// TIA Portal V18 program export: 1 tag tables, 0 data types, 0 data blocks, 6 code blocks (in call order from the OBs), 0 instance data blocks

VAR_GLOBAL   // PLC tag table "Default tag table"
   convRight AT %I0.0 : Bool;
   convLeft AT %I0.1 : Bool;
   manualMode AT %Q0.2 : Bool;
   automaticMode AT %Q0.3 : Bool;
END_VAR

ORGANIZATION_BLOCK "Main"   // OB1, LAD, ProgramCycle
TITLE = "Main Program Sweep (Cycle)"
{ S7_Optimized_Access := 'TRUE' }
VERSION : 0.1
// stored: AutoNumber true, IsIECCheckEnabled true, SetENOAutomatically false
   VAR_INPUT
      Initial_Call : Bool;   // Initial call of this OB
      Remanence : Bool;   // =True, if remanent data are available
   END_VAR
BEGIN
END_ORGANIZATION_BLOCK

FUNCTION_BLOCK "Conveyor"   // FB2, FBD
{ S7_Optimized_Access := 'TRUE' }
AUTHOR : dda
VERSION : 0.1
// stored: AutoNumber true, IsIECCheckEnabled true, IsRetainMemResEnabled false, MemoryReserve 100, SetENOAutomatically true, UDAEnableTagReadback false
   VAR_INPUT
      automaticMode { ExternalAccessible := 'False'; ExternalVisible := 'False'; ExternalWritable := 'False'} : Bool;
      manualMode { ExternalAccessible := 'False'; ExternalVisible := 'False'; ExternalWritable := 'False'} : Bool;
      jogRight { ExternalAccessible := 'False'; ExternalVisible := 'False'; ExternalWritable := 'False'} : Bool;
      run { ExternalAccessible := 'False'; ExternalVisible := 'False'; ExternalWritable := 'False'} : Bool;
   END_VAR
   VAR_OUTPUT
      conveyorRight { ExternalAccessible := 'False'; ExternalVisible := 'False'; ExternalWritable := 'False'} : Bool;
      conveyorLeft { ExternalAccessible := 'False'; ExternalVisible := 'False'; ExternalWritable := 'False'} : Bool;
   END_VAR
   VAR
      statRequest { ExternalAccessible := 'False'; ExternalVisible := 'False'; ExternalWritable := 'False'} : Bool;
      statRelease { ExternalAccessible := 'False'; ExternalVisible := 'False'; ExternalWritable := 'False'} : Bool;
   END_VAR
BEGIN

REGION Network 1 (SCL)
   // functionality: conveyor
   //
END_REGION

REGION Network 2
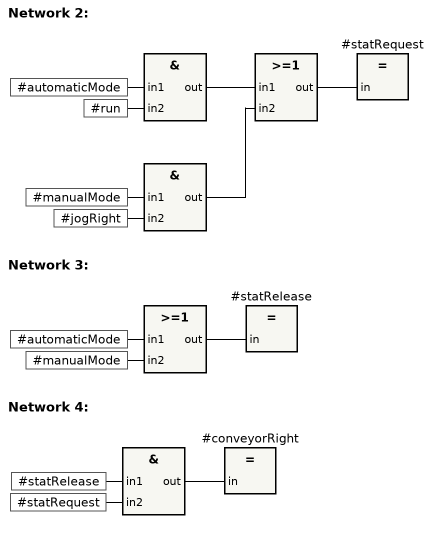
   #statRequest := (#automaticMode AND #run) OR (#manualMode AND #jogRight);
END_REGION

REGION Network 3
   #statRelease := #automaticMode OR #manualMode;
END_REGION

REGION Network 4
   #conveyorRight := #statRelease AND #statRequest;
END_REGION
END_FUNCTION_BLOCK

FUNCTION_BLOCK "Seqencer"   // FB4, GRAPH
AUTHOR : dda
VERSION : 0.1
// stored: AcknowledgeErrorsRequired true, AutoNumber true, GraphVersion 6.0, InitialValuesAcquisition false, IsIECCheckEnabled true, LanguageInNetworks FBD, LockOperatingMode false, PermanentILProcessingInMANMode false, SetENOAutomatically true, SkipSteps false, UDAEnableTagReadback false, WithAlarmHandling true
   // inherited from GRAPH_BASE
   VAR
      OFF_SQ_BASE : Bool;
   END_VAR
   VAR_INPUT
      OFF_SQ { ExternalWritable := 'False'} : Bool := false;   // Turn sequence off
      INIT_SQ { ExternalWritable := 'False'} : Bool := false;   // Set sequence to initial state
      ACK_EF { ExternalWritable := 'False'} : Bool := false;   // Acknowledge all errors and faults
      REG_EF { ExternalWritable := 'False'} : Bool := false;   // Register all errors and faults
      ACK_S { ExternalWritable := 'False'} : Bool := false;   // Acknowledge step indicated in S_NO
      REG_S { ExternalWritable := 'False'} : Bool := false;   // Register the step indicated in S_NO
      HALT_SQ { ExternalWritable := 'False'} : Bool := false;   // Halt sequence immediately
      HALT_TM { ExternalWritable := 'False'} : Bool := false;   // Halt timers immediately
      ZERO_OP { ExternalWritable := 'False'} : Bool := false;   // Set all operands assigned with N, L, D to 0
      EN_IL { ExternalWritable := 'False'} : Bool := false;   // Enable interlocks
      EN_SV { ExternalWritable := 'False'} : Bool := false;   // Activate supervision processing
      EN_ACKREQ { ExternalWritable := 'False'} : Bool := false;   // Activate mandatory acknowledgment
      EN_SSKIP { ExternalWritable := 'False'} : Bool := false;   // Enable "Skip step"
      DISP_SACT { ExternalWritable := 'False'} : Bool := false;   // Display active steps only
      DISP_SEF { ExternalWritable := 'False'} : Bool := false;   // Display only steps with errors and disrupted steps
      DISP_SALL { ExternalWritable := 'False'} : Bool := false;   // Display all steps
      S_PREV { ExternalWritable := 'False'} : Bool := false;   // Output previous step in parameter S_NO
      S_NEXT { ExternalWritable := 'False'} : Bool := false;   // Indicate next step in parameter S_NO
      SW_AUTO { ExternalWritable := 'False'} : Bool := false;   // Automatic mode
      SW_TAP { ExternalWritable := 'False'} : Bool := false;   // Semiautomatic/switch with transition
      SW_TOP { ExternalWritable := 'False'} : Bool := false;   // Semiautomatic/ignore transition
      SW_MAN { ExternalWritable := 'False'} : Bool := false;   // Manual mode
      S_SEL { ExternalWritable := 'False'} : Int := 0;   // Select step to be output to S_NO
      S_SELOK { ExternalWritable := 'False'} : Bool := false;   // Enter value from S_SEL in S_NO
      S_ON { ExternalWritable := 'False'} : Bool := false;   // Activate step indicated in S_NO
      S_OFF { ExternalWritable := 'False'} : Bool := false;   // Disable step indicated in S_NO
      T_PREV { ExternalWritable := 'False'} : Bool := false;   // Display previous transition in T_NO
      T_NEXT { ExternalWritable := 'False'} : Bool := false;   // Display next transition at parameter T_NO
      T_PUSH { ExternalWritable := 'False'} : Bool := false;   // Enable transition to switch in semi automatic mode
      EN_LMODE { ExternalWritable := 'False'} : Bool := false;   // Activate learning mode
      RESET_CRIT { ExternalWritable := 'False'} : Bool := false;   // Reset all initial values recorded for interlocks and transitions
      startButton : Bool;
      lightBeam1 : Bool;
      lightBeam2 : Bool;
      lightBeam3 : Bool;
      robotArmDown : Bool;
      robotOnStation : Bool;
      robotOnMagazine : Bool;
      mySupervision : Bool;
   END_VAR
   VAR_OUTPUT
      S_NO { ExternalWritable := 'False'} : Int := 0;   // Step number
      S_MORE { ExternalWritable := 'False'} : Bool := false;   // More steps are available and can be shown in S_NO
      S_ACTIVE { ExternalWritable := 'False'} : Bool := false;   // Step indicated in S_NO is active
      S_TIME { ExternalWritable := 'False'} : Time := T#0ms;   // Step activation time
      S_TIMEOK { ExternalWritable := 'False'} : Time := T#0ms;   // No error in step activation time
      S_CRITLOC { ExternalWritable := 'False'} : DWord := 16#0;   // Interlock criteria bits
      S_CRITLOCERR { ExternalWritable := 'False'} : DWord := 16#0;   // Interlock criteria bits for event L1
      S_STATE { ExternalWritable := 'False'} : Word := 16#0;   // Step state bits
      T_NO { ExternalWritable := 'False'} : Int := 0;   // Transition number
      T_MORE { ExternalWritable := 'False'} : Bool := false;   // More valid transitions available for display
      T_CRIT { ExternalWritable := 'False'} : DWord := 16#0;   // Transition criteria bits
      T_CRITOLD { ExternalWritable := 'False'} : DWord := 16#0;   // Transition criteria bits from last cycle
      T_CRITFLT { ExternalWritable := 'False'} : DWord := 16#0;   // Transition criteria bits for event V1
      ERROR { ExternalWritable := 'False'} : Bool := false;   // Interlock group error
      FAULT { ExternalWritable := 'False'} : Bool := false;   // Supervision group error
      ERR_FLT { ExternalWritable := 'False'} : Bool := false;   // Interlock or supervision group error
      SQ_ISOFF { ExternalWritable := 'False'} : Bool := false;   // Sequence is off (no step active)
      SQ_HALTED { ExternalWritable := 'False'} : Bool := false;   // Sequence halted
      TM_HALTED { ExternalWritable := 'False'} : Bool := false;   // Timers halted
      OP_ZEROED { ExternalWritable := 'False'} : Bool := false;   // All the operands assigned with N, L, D are set to 0
      IL_ENABLED { ExternalWritable := 'False'} : Bool := false;   // Interlocks are active
      SV_ENABLED { ExternalWritable := 'False'} : Bool := false;   // Supervision processing activated
      ACKREQ_ENABLED { ExternalWritable := 'False'} : Bool := false;   // Mandatory acknowledgment activated
      SSKIP_ENABLED { ExternalWritable := 'False'} : Bool := false;   // Skip steps activated
      SACT_DISP { ExternalWritable := 'False'} : Bool := false;   // Display active steps only
      SEF_DISP { ExternalWritable := 'False'} : Bool := false;   // Display only steps with errors or disrupted steps
      SALL_DISP { ExternalWritable := 'False'} : Bool := false;   // Display all steps
      AUTO_ON { ExternalWritable := 'False'} : Bool := false;   // Automatic mode is active
      TAP_ON { ExternalWritable := 'False'} : Bool := false;   // Semiautomatic mode/step with transition enabled
      TOP_ON { ExternalWritable := 'False'} : Bool := false;   // Semiautomatic mode/ignore transition enabled
      MAN_ON { ExternalWritable := 'False'} : Bool := false;   // Manual mode is active
      LMODE_ENABLED { ExternalWritable := 'False'} : Bool := false;   // Learning mode is active
      partInPos1 { ExternalAccessible := 'False'; ExternalVisible := 'False'; ExternalWritable := 'False'} : Bool;
      partInPos2 { ExternalAccessible := 'False'; ExternalVisible := 'False'; ExternalWritable := 'False'} : Bool;
      partInPos3 { ExternalAccessible := 'False'; ExternalVisible := 'False'; ExternalWritable := 'False'} : Bool;
      startConv { ExternalAccessible := 'False'; ExternalVisible := 'False'; ExternalWritable := 'False'} : Bool;
      automaticMode { ExternalAccessible := 'False'; ExternalVisible := 'False'; ExternalWritable := 'False'} : Bool;
      robotFill { ExternalAccessible := 'False'; ExternalVisible := 'False'; ExternalWritable := 'False'} : Bool;
      robotGoToMagazine { ExternalAccessible := 'False'; ExternalVisible := 'False'; ExternalWritable := 'False'} : Bool;
      robotGoToStation { ExternalAccessible := 'False'; ExternalVisible := 'False'; ExternalWritable := 'False'} : Bool;
   END_VAR
   VAR
      statLightbeam3Fal { ExternalAccessible := 'False'; ExternalVisible := 'False'; ExternalWritable := 'False'} : Bool;
      statMemoryTag { ExternalAccessible := 'False'; ExternalVisible := 'False'; ExternalWritable := 'False'} : Bool;
   END_VAR
BEGIN
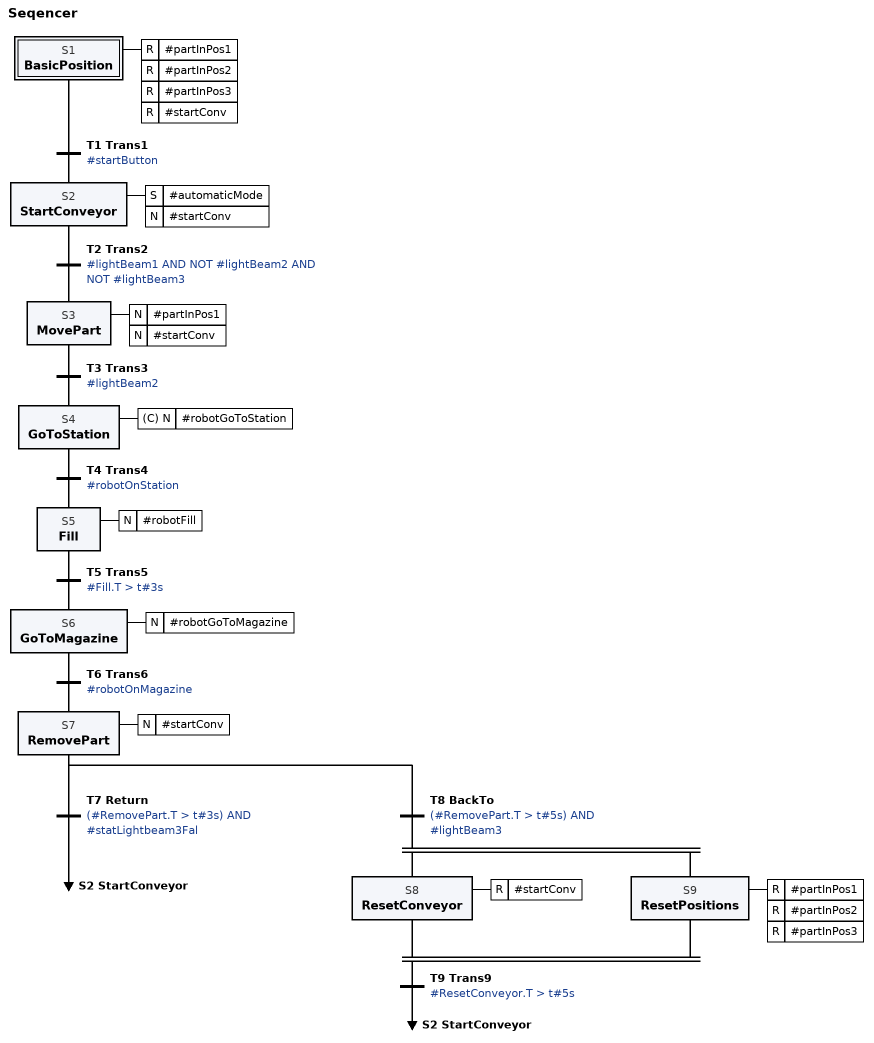
   // sequencer 1
   INITIAL_STEP BasicPosition:   // S1, max time T#10S, warning time T#7S
      supervision V := (#StartConveyor.T > t#10ms) AND (#StartConveyor.U > t#10ms);
              R    #partInPos1
              R    #partInPos2
              R    #partInPos3
              R    #startConv
   END_STEP
   TRANSITION Trans1 FROM BasicPosition TO StartConveyor   // T1
      := #startButton;
   END_TRANSITION
   STEP StartConveyor:   // S2, max time T#10S, warning time T#7S
              S    #automaticMode
              N    #startConv
   END_STEP
   TRANSITION Trans2 FROM StartConveyor TO MovePart   // T2
      := #lightBeam1 AND NOT #lightBeam2 AND NOT #lightBeam3;
   END_TRANSITION
   STEP MovePart:   // S3, max time T#10S, warning time T#7S
              N    #partInPos1
              N    #startConv
   END_STEP
   TRANSITION Trans3 FROM MovePart TO GoToStation   // T3
      := #lightBeam2;
   END_TRANSITION
   STEP GoToStation:   // S4, max time T#10S, warning time T#7S
      interlock C := NOT #robotArmDown;
      (C)     N    #robotGoToStation
   END_STEP
   TRANSITION Trans4 FROM GoToStation TO Fill   // T4
      := #robotOnStation;
   END_TRANSITION
   STEP Fill:   // S5, max time T#10S, warning time T#7S
              N    #robotFill
   END_STEP
   TRANSITION Trans5 FROM Fill TO GoToMagazine   // T5
      := #Fill.T > t#3s;
   END_TRANSITION
   STEP GoToMagazine:   // S6, max time T#10S, warning time T#7S
              N    #robotGoToMagazine
   END_STEP
   TRANSITION Trans6 FROM GoToMagazine TO RemovePart   // T6
      := #robotOnMagazine;
   END_TRANSITION
   STEP RemovePart:   // S7, max time T#10S, warning time T#7S
      supervision V := (#RemovePart.T < #RemovePart.T_MAX) AND (#RemovePart.T > #RemovePart.T_WARN);
              N    #startConv
   END_STEP
   TRANSITION "Return" FROM RemovePart TO StartConveyor   // T7, jump
      := (#RemovePart.T > t#3s) AND #statLightbeam3Fal;
   END_TRANSITION
   TRANSITION BackTo FROM RemovePart TO (ResetConveyor, ResetPositions)   // T8
      := (#RemovePart.T > t#5s) AND #lightBeam3;
   END_TRANSITION
   STEP ResetConveyor:   // S8, max time T#10S, warning time T#7S
              R    #startConv
   END_STEP
   STEP ResetPositions:   // S9, max time T#10S, warning time T#7S
      interlock C := #ResetPositions.T > #ResetPositions.T_MAX;
              R    #partInPos1
              R    #partInPos2
              R    #partInPos3
   END_STEP
   TRANSITION Trans9 FROM (ResetConveyor, ResetPositions) TO StartConveyor   // T9, jump
      := #ResetConveyor.T > t#5s;
   END_TRANSITION
END_FUNCTION_BLOCK

FUNCTION_BLOCK "Simulation"   // FB1, FBD
TITLE = Simulation
{ S7_Optimized_Access := 'TRUE' }
AUTHOR : dda
VERSION : 0.1
// Simulate machine behaviour
// stored: AutoNumber true, IsIECCheckEnabled true, IsRetainMemResEnabled false, MemoryReserve 100, SetENOAutomatically true, UDAEnableTagReadback false
   VAR_INPUT
      moveUp { ExternalAccessible := 'False'; ExternalVisible := 'False'; ExternalWritable := 'False'} : Bool;
      moveDown { ExternalAccessible := 'False'; ExternalVisible := 'False'; ExternalWritable := 'False'} : Bool;
      MoveLeft { ExternalAccessible := 'False'; ExternalVisible := 'False'; ExternalWritable := 'False'} : Bool;
      moveRight { ExternalAccessible := 'False'; ExternalVisible := 'False'; ExternalWritable := 'False'} : Bool;
      runConveyor { ExternalAccessible := 'False'; ExternalVisible := 'False'; ExternalWritable := 'False'} : Bool;
      engineBroken { ExternalAccessible := 'False'; ExternalVisible := 'False'; ExternalWritable := 'False'} : Bool;
      robotGoToStation { ExternalAccessible := 'False'; ExternalVisible := 'False'; ExternalWritable := 'False'} : Bool;
      robotGoToMagazine { ExternalAccessible := 'False'; ExternalVisible := 'False'; ExternalWritable := 'False'} : Bool;
   END_VAR
   VAR_OUTPUT
      xPosition { ExternalAccessible := 'False'; ExternalVisible := 'False'; ExternalWritable := 'False'} : Int;
      yPosition { ExternalAccessible := 'False'; ExternalVisible := 'False'; ExternalWritable := 'False'} : Int;
      lightBeam1 { ExternalAccessible := 'False'; ExternalVisible := 'False'; ExternalWritable := 'False'} : Bool;
      lightBeam2 { ExternalAccessible := 'False'; ExternalVisible := 'False'; ExternalWritable := 'False'} : Bool;
      lightBeam3 { ExternalAccessible := 'False'; ExternalVisible := 'False'; ExternalWritable := 'False'} : Bool;
      robotPosHMI { ExternalAccessible := 'False'; ExternalVisible := 'False'; ExternalWritable := 'False'} : Int;
      robotHasChip { ExternalAccessible := 'False'; ExternalVisible := 'False'; ExternalWritable := 'False'} : Bool;
   END_VAR
   VAR
      instTimerSimulate { ExternalAccessible := 'False'; ExternalVisible := 'False'; ExternalWritable := 'False'; S7_SetPoint := 'True'} : TON_TIME;
      statSimulate { ExternalAccessible := 'False'; ExternalVisible := 'False'; ExternalWritable := 'False'} : Bool;
      StatPositionConveyor { ExternalAccessible := 'False'; ExternalVisible := 'False'; ExternalWritable := 'False'} : Int;
      statRobotHasChip { ExternalAccessible := 'False'; ExternalVisible := 'False'; ExternalWritable := 'False'} : Bool;
      statRobotPosHMI { ExternalAccessible := 'False'; ExternalVisible := 'False'; ExternalWritable := 'False'} : Int;
   END_VAR
   VAR_TEMP
      tempLB1 : Bool;
      tempLB2 : Bool;
      tempLB3 : Bool;
   END_VAR
   VAR CONSTANT
      SIMULATION_TIME : Time := T#10ms;
   END_VAR
BEGIN

REGION Network 1 (SCL)
   // Титульные комменты для блока
   // 
   // 22.12.2023
END_REGION

REGION Network 2: trigger simulation step
   // set bit one cycle every 10 ms
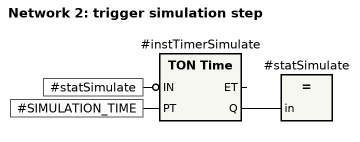
   #instTimerSimulate(IN := NOT #statSimulate, PT := #SIMULATION_TIME);   // TON
   #statSimulate := #instTimerSimulate.Q;
END_REGION

REGION Network 3 (SCL): Simulation step
   IF (#statSimulate = TRUE) AND (NOT #engineBroken) THEN
     // move robot
     IF #moveUp = TRUE THEN
       #yPosition += 1;
     END_IF;
     IF #moveDown = TRUE THEN
       #yPosition -= 1;
     END_IF;
     IF #MoveLeft = TRUE THEN
       #xPosition += 1;
     END_IF;
     IF #moveRight = TRUE THEN
       #xPosition -= 1;
     END_IF;
     // move conveyor
     IF (#StatPositionConveyor > 800) THEN
       #StatPositionConveyor := 0;
     ELSIF (#runConveyor = TRUE) THEN
       #StatPositionConveyor += 1;
     END_IF;
   END_IF;

   // for S7-300 / S7-400
   #tempLB1 := FALSE;
   #tempLB2 := FALSE;
   #tempLB3 := FALSE;

   // assign lightbeams
   CASE #StatPositionConveyor OF
     30..60:
       #tempLB1 := TRUE;
     500..530:
       #tempLB2 := TRUE;
     700..800:
       #tempLB3 := TRUE;

     ELSE   // Statement section ELSE
       ;
   END_CASE;

   #lightBeam1 := #tempLB1;
   #lightBeam2 := #tempLB2;
   #lightBeam3 := #tempLB3;

   // Calculate data for display of robot in HMI
   IF (#xPosition = 100)
   THEN
     #statRobotPosHMI := #yPosition;
   ELSE
     #statRobotPosHMI := 100;
   END_IF;
END_REGION
END_FUNCTION_BLOCK

FUNCTION_BLOCK "ExtensionToGRAPH"
{ S7_Optimized_Access := 'TRUE' }
AUTHOR : dda
VERSION : 0.1
   VAR_IN_OUT 
      extRTData {InstructionName := 'G7_RTDataPlus_V6'; LibVersion := '1.0'} : G7_RTDataPlus_V6;
      extG7T {InstructionName := 'G7_TransitionPlus_V6'; LibVersion := '1.0'} : Array[*] of G7_TransitionPlus_V6;
      extG7S {InstructionName := 'G7_StepPlus_V6'; LibVersion := '1.0'} : Array[*] of G7_StepPlus_V6;
      extG7Arrays : Array[*] of USInt;
   END_VAR

   VAR 
      statLowerG7T { ExternalAccessible := 'False'; ExternalVisible := 'False'; ExternalWritable := 'False'} : DInt;
      statUpperG7T { ExternalAccessible := 'False'; ExternalVisible := 'False'; ExternalWritable := 'False'} : DInt;
      statLowerG7S { ExternalAccessible := 'False'; ExternalVisible := 'False'; ExternalWritable := 'False'} : DInt;
      statUpperG7S { ExternalAccessible := 'False'; ExternalVisible := 'False'; ExternalWritable := 'False'} : DInt;
      statUserTransitionNumber : Int;
      statUserStepNumber : Int;
      statUserActiveSteps : USInt;
      statUserSatisfiedTrans : USInt;
   END_VAR

   VAR_TEMP 
      tempG7TIndex : DInt;
      tempG7SIndex : DInt;
   END_VAR


BEGIN
	// Functionality: extension functionality for iterative acces to Graph 
	// variables and invisible GraphStatusVariables.
	// 
	
	REGION ReadArrayBoundaries
	  // Read ArrayBoundaries of predefinedGreph-Array's
	  // 
	  #statLowerG7T := LOWER_BOUND(ARR := #extG7T, DIM := 1);
	  #statUpperG7T := UPPER_BOUND(ARR := #extG7T, DIM := 1);
	  
	  #statLowerG7S := LOWER_BOUND(ARR := #extG7S, DIM := 1);
	  #statUpperG7S := UPPER_BOUND(ARR := #extG7S, DIM := 1);
	  
	  
	END_REGION
	
	
	REGION IterrativeTransitionAcces
	  // Example: As a programmer I want to check whether a specific transation
	  // number (e.g. asked via HMI-Panel) is available in the Graph block.
	  // 
	  
	  FOR #tempG7TIndex := #statLowerG7T TO #statUpperG7T  BY 1 DO
	    ;
	    IF (#extG7T[#tempG7TIndex].TNO = #statUserTransitionNumber)
	    THEN
	      ;
	      // do any action
	    END_IF;
	  END_FOR;
	  
	  
	END_REGION
	
	REGION IterrativeStepAcces
	  // Example: As a programmer I want to check whether a specific step
	  // number (e.g. asked via HMI-Panel) is available in the Graph block.
	  // 
	  
	  FOR #tempG7SIndex := #statLowerG7S TO #statUpperG7S BY 1 DO
	    ;
	    IF (#extG7S[#tempG7SIndex].SNO = #statUserStepNumber)
	    THEN
	      ;
	      // do any action
	    END_IF;
	  END_FOR;
	  
	  
	END_REGION
	
	REGION ReadGraphStatusVariables
	  
	  #statUserActiveSteps := #extG7Arrays[#extRTData.OFFSETS.SAX_OFFSET] - 1;
	  
	  #statUserSatisfiedTrans := #extG7Arrays[#extRTData.OFFSETS.TTX_OFFSET] - 1;
	  
	END_REGION
	
	
	
END_FUNCTION_BLOCK

FUNCTION_BLOCK "Robot"
{ S7_Optimized_Access := 'TRUE' }
AUTHOR : dda
VERSION : 0.1
   VAR_INPUT 
      goToMagazine { ExternalAccessible := 'False'; ExternalVisible := 'False'; ExternalWritable := 'False'} : Bool;
      goToStation { ExternalAccessible := 'False'; ExternalVisible := 'False'; ExternalWritable := 'False'} : Bool;
      fill { ExternalAccessible := 'False'; ExternalVisible := 'False'; ExternalWritable := 'False'} : Bool;
      xPosition { ExternalAccessible := 'False'; ExternalVisible := 'False'; ExternalWritable := 'False'} : Int;
      yPosition { ExternalAccessible := 'False'; ExternalVisible := 'False'; ExternalWritable := 'False'} : Int;
   END_VAR

   VAR_OUTPUT 
      pressingNut { ExternalAccessible := 'False'; ExternalVisible := 'False'; ExternalWritable := 'False'} : Bool;
      moveUp { ExternalAccessible := 'False'; ExternalVisible := 'False'; ExternalWritable := 'False'} : Bool;
      moveDown { ExternalAccessible := 'False'; ExternalVisible := 'False'; ExternalWritable := 'False'} : Bool;
      moveLeft { ExternalAccessible := 'False'; ExternalVisible := 'False'; ExternalWritable := 'False'} : Bool;
      isOnStation { ExternalAccessible := 'False'; ExternalVisible := 'False'; ExternalWritable := 'False'} : Bool;
      isOnMagazine { ExternalAccessible := 'False'; ExternalVisible := 'False'; ExternalWritable := 'False'} : Bool;
      moveRight { ExternalAccessible := 'False'; ExternalVisible := 'False'; ExternalWritable := 'False'} : Bool;
   END_VAR

   VAR 
      statMoveUp { ExternalAccessible := 'False'; ExternalVisible := 'False'; ExternalWritable := 'False'} : Bool;
      statMoveDown { ExternalAccessible := 'False'; ExternalVisible := 'False'; ExternalWritable := 'False'} : Bool;
      statMoveLeft { ExternalAccessible := 'False'; ExternalVisible := 'False'; ExternalWritable := 'False'} : Bool;
      statMoveRight { ExternalAccessible := 'False'; ExternalVisible := 'False'; ExternalWritable := 'False'} : Bool;
      statIsOnMagazine { ExternalAccessible := 'False'; ExternalVisible := 'False'; ExternalWritable := 'False'} : Bool;
      statPressingNut { ExternalAccessible := 'False'; ExternalVisible := 'False'; ExternalWritable := 'False'} : Bool;
      statGoToStation { ExternalAccessible := 'False'; ExternalVisible := 'False'; ExternalWritable := 'False'} : Bool;
      statIsOnStation { ExternalAccessible := 'False'; ExternalVisible := 'False'; ExternalWritable := 'False'} : Bool;
      statRobot { ExternalAccessible := 'False'; ExternalVisible := 'False'; ExternalWritable := 'False'} : Int;
   END_VAR

   VAR_TEMP 
      tempYPosition : Int;
      tempXPosition : Int;
   END_VAR

   VAR CONSTANT 
      ARM_UP : Int := 1;   // object arrived position 1
      DIRECTION_RIGHT : Int := 6;
      OBJECT_FILL : Int := 4;   // object arrived position 2 and not filled
      DIRECTION_LEFT : Int := 2;
      ARM_DOWN : Int := 3;   // object arrived position 2 and Filled
      ARM_UP_BACK : Int := 5;
      ARM_DOWN_BACK : Int := 7;
      IDLE : Int := 0;
   END_VAR


BEGIN
	// functionality: Robot
	// 
	
	// read inputs
	#tempYPosition := #yPosition;
	#tempXPosition := #xPosition;
	
	CASE #statRobot OF
	    // robot on magazine
	  #IDLE:
	    #statMoveDown := FALSE;
	    #statIsOnMagazine := FALSE;
	    IF (#goToStation = TRUE) THEN
	      #statRobot := #ARM_UP;
	    END_IF;
	    
	    // robot move up
	  #ARM_UP:
	    #statMoveDown := FALSE;
	    #statMoveUp := TRUE;
	    IF (#tempYPosition = 100) THEN
	      #statRobot := #ARM_UP;
	    END_IF;
	    
	    // robot moves to the left direction  
	  #DIRECTION_LEFT:
	    #statMoveUp := FALSE;
	    #statMoveLeft := TRUE;
	    IF (#tempXPosition = 100) THEN
	      #statRobot := #ARM_DOWN;
	    END_IF;
	    
	    // robot moves down
	  #ARM_DOWN:
	    #statMoveLeft := FALSE;
	    #statMoveDown := TRUE;
	    IF (#tempYPosition = 0) THEN
	      #statIsOnStation := TRUE;
	      #statRobot := #OBJECT_FILL;
	    END_IF;
	    
	    // fill
	  #OBJECT_FILL:
	    #statMoveDown := FALSE;
	    #statIsOnStation := FALSE;
	    #statPressingNut := #fill;
	    IF (#goToMagazine = TRUE) THEN
	      #statRobot := #ARM_UP_BACK;
	    END_IF;
	    
	    // robot moves up
	  #ARM_UP_BACK:
	    #statMoveUp := true;
	    #statPressingNut := FALSE;
	    IF (#tempYPosition = 100) THEN
	      #statRobot := #DIRECTION_RIGHT;
	    END_IF;
	    
	    // robot moves to the right direction
	  #DIRECTION_RIGHT:
	    #statMoveUp := FALSE;
	    #statMoveRight := TRUE;
	    IF (#tempXPosition = 0) THEN
	      #statRobot := #ARM_DOWN_BACK;
	    END_IF;
	    
	    // robot moves down back to magazine
	  #ARM_DOWN_BACK:
	    #statMoveRight := FALSE;
	    #statMoveDown := TRUE;
	    IF (#tempYPosition = 0) THEN
	      #statIsOnMagazine := TRUE;
	      #statRobot := #IDLE;
	    END_IF;
	    
	  ELSE
	    ;
	END_CASE;
	
	// write outputs
	#moveUp := #statMoveUp;
	#moveDown := #statMoveDown;
	#moveLeft := #statMoveLeft;
	#moveRight := #statMoveRight;
	#isOnMagazine := #statIsOnMagazine;
	#isOnStation := #statIsOnStation;
	#pressingNut := #statPressingNut;
	      
	      
	    
	      
	        
	      
	      
	
END_FUNCTION_BLOCK
